VAR_GLOBAL // INPUTS
    ivar_g_inp AT %I*: DINT;
END_VAR

(* stored: ProductVersion 3.1.0.18, Version 1.1.0.1 *)
